FUNCTION_BLOCK T_Gripper EXTENDS T_NamedBase IMPLEMENTS I_Gripper
VAR
END_VAR

END_FUNCTION_BLOCK

(* stored: Version 1.1.0.1, ProductVersion 3.1.4024.12
   POU T_Gripper: Id {f66baa9a-c4d1-4cbd-b572-4fc9913db1d8}, SpecialFunc None *)
